TEXTLIST TextList_RTR_errorid
  0 = 'no_error'
  1 = 'not_connected'
  2 = 'invalid_state'
  4 = 'cmd_timeout'
  5 = 'unknown_error'
  6 = 'Drive_not_ready_for_operation'
  666 = 'emergency_error'
  3 = 'break_exceeded_timeout'
  7 = 'roll_unclamped'
   = ''
END_TEXTLIST

(* stored: Version 1.1.0.1, ProductVersion 3.1.4024.11
   TextList TextList_RTR_errorid: Id {645fa0b6-b988-4bd0-9498-1a71a062aa61} *)
